// TIA Portal project "AWL LIBRO 8" (V11)

(* hardware
DEVICE "S7300/ET200 station_1"  SIMATIC 300-Station
   slot 0: "Perfil soporte_0"  Rail  6ES7 390-1***0-0AA0
   slot 2: "PLC_1"  CPU 313C-2 DP  6ES7 313-6CF03-0AB0  V2.6
      slot 0: "Interfaz MPI_1"  MPI
      slot 1: "Interfaz DP_1"  DP
      slot 2: "DI16/DO16_1"  DI16/DO16
      slot 4: "Contaje_1"  Counter
*)

// ===== PLC "PLC_1"  CPU 313C-2 DP =====

VAR_GLOBAL   // PLC tag table "Tabla de variables estándar"
   "PRESELECCION" AT %E0.0 : Bool;
   "EJECUCION" AT %E0.1 : Bool;
   "LED BOMBA 1" AT %A0.0 : Bool;
   "LED BOMBA 2" AT %A0.1 : Bool;
   "LED BOMBA 3" AT %A0.2 : Bool;
   "LED BOMBA 4" AT %A0.3 : Bool;
   "EMERGENCIA" AT %E0.2 : Bool;
   "BOMBA 1 FUNCIONANDO" AT %A0.4 : Bool;
   "BOMBA 2 FUNCIONANDO" AT %A0.5 : Bool;
   "BOMBA 3 FUNCIONANDO" AT %A0.6 : Bool;
   "BOMBA 4 FUNCIONANDO" AT %A0.7 : Bool;
   "CONTADOR" AT %MW0 : Int;
   "SALIDAS" AT %AB0 : Byte;
   "T0" AT %T0 : Timer;
   "Tag_1" AT %E0.7 : Bool;
   "Tag_2" AT %A1.0 : Bool;
   "Tag_3" AT %M10.0 : Bool;
   "Tag_4" AT %M10.2 : Bool;
   "Tag_5" AT %M10.1 : Bool;
   "Tag_6" AT %M10.3 : Bool;
   "Tag_7" AT %MB10 : Byte;
   "Tag_8" AT %M0.4 : Bool;
   "Tag_9" AT %M0.5 : Bool;
   "Tag_10" AT %M10.5 : Bool;
   "Tag_11" AT %M10.4 : Bool;
   "Tag_12" AT %M10.6 : Bool;
   "Tag_13" AT %M10.7 : Bool;
   "Tag_14" AT %M100.5 : Bool;
   "Tag_15" AT %M1.2 : Bool;
END_VAR

DATA_BLOCK "F Y B"   // DB1
{ S7_Optimized_Access := 'FALSE' }
VERSION : 0.1
   VAR
      F0 : Bool;
      F1 : Bool;
      F2 : Bool;
      F3 : Bool;
      F4 : Bool;
      F5 : Bool;
      F6 : Bool;
      F7 : Bool;
      F8 : Bool;
      B0 : Bool;
      B1 : Bool;
      B2 : Bool;
      B3 : Bool;
      B4 : Bool;
      B5 : Bool;
      B6 : Bool;
      B7 : Bool;
   END_VAR
BEGIN
END_DATA_BLOCK

ORGANIZATION_BLOCK "Main"   // OB1, STL
TITLE = EJERCIICO 8. / "Main Program Sweep (Cycle)"
{ S7_Optimized_Access := 'FALSE' }
VERSION : 0.1
   VAR_TEMP
      OB1_EV_CLASS : Byte;   // Bits 0-3 = 1 (Coming event), Bits 4-7 = 1 (Event class 1)
      OB1_SCAN_1 : Byte;   // 1 (Cold restart scan 1 of OB 1), 3 (Scan 2-n of OB 1)
      OB1_PRIORITY : Byte;   // Priority of OB Execution
      OB1_OB_NUMBR : Byte;   // 1 (Organization block 1, OB1)
      OB1_RESERVED_1 : Byte;   // Reserved for system
      OB1_RESERVED_2 : Byte;   // Reserved for system
      OB1_PREV_CYCLE : Int;   // Cycle time of previous OB1 scan (milliseconds)
      OB1_MIN_CYCLE : Int;   // Minimum cycle time of OB1 (milliseconds)
      OB1_MAX_CYCLE : Int;   // Maximum cycle time of OB1 (milliseconds)
      OB1_DATE_TIME : Date_And_Time;   // Date and time OB1 started
   END_VAR
BEGIN
END_ORGANIZATION_BLOCK